PROGRAM ExtMode_Init
VAR
	iSTEP : INT:= 0;
	Pulse1			: TP; //for drive_on pulse
	Pulse2			: TP; //for ext_start pulse
	Pulse3			: TP;
	Pulse4			: TP;
	
	rInit			: R_TRIG;   // latch one press
	bInitLatch		: BOOL := FALSE;
	//bExtOK			: BOOL := IO_KUKA.bEXT_mode ;
	   
    rStep10       : R_TRIG;   // "step 10 entered" one-shot
    rStep30       : R_TRIG;   // "step 30 entered" one-shot
    tonPeri    : TON;      // wait for $PERI_RDY
    tonStart   : TON;      // wait for $PRO_ACT
    tPulse     : TIME := T#300MS;
    tPeriTO    : TIME := T#10S;
    tStartTO   : TIME := T#10S;
	
	
	
END_VAR


//// ================  Edges  ================
////rInit(CLK := IO_KUKA.Init_Cmd);
//rStep10(CLK := (iSTEP =10));
//rStep30(CLK := (iSTEP =30));

//IF IO_KUKA.Init_Cmd AND IO_KUKA.bEXT_mode = TRUE THEN
//	bInitLatch := TRUE;
//END_IF

//IF iSTEP <> 0 THEN
//	IO_control.bMove_enable := TRUE;   // $MOVE_ENABLE = 1
//    IO_control.bDrive_off   := FALSE;  // $DRIVES_OFF = 0
//	IO_control.bIO_Act      := TRUE;   // your "Activate interface" bit
//END_IF


//// ================  Machine state  ================
//CASE iSTEP OF
//	// ================  0 : idle  ================
//	0:	
//		IO_control.bDrive_on  	:= FALSE;
//  	 	IO_control.bExt_start 	:= FALSE;
//    	IO_control.bConf_msg  	:= FALSE;
//  		IO_control.bMove_enable := FALSE;
//    	IO_control.bIO_Act      := FALSE;
//   		IO_control.bDrive_off   := FALSE;
		
//		IF bInitLatch THEN
//			iSTEP := 10;
//		END_IF
		
//	// ================  10 : pulse drives_on, start wait for peri_rdy  ================
//	10:	
//		Pulse1(IN := rStep10.Q, PT := tPulse);
//		IO_control.bDrive_on := Pulse1.Q;
		
//		IF rStep10.Q THEN
//			tonPeri(IN := TRUE, PT := tPeriTO);
//			iSTEP := 20;
//		END_IF

		
//	// ================  20 : pwait for peri_rdy, conf_mess follows stopmess  ================
//	20:	
//		IO_control.bConf_msg := IO_KUKA.bStopmess;
		
//		IF IO_KUKA.bPeri_ready THEN
//			tonPeri(IN := FALSE);
//			iSTEP := 30;
//		ELSE
//			bInitLatch := FALSE;
//        	tonPeri(IN := FALSE);
//        	iSTEP := 0;
//		END_IF
	

//	// ================  30 : when no stopmess, pulse ext_start and wait Pro_act  ================
//	30:
//		IO_control.bConf_msg := IO_KUKA.bStopmess;
		
//		IF NOT IO_KUKA.bStopmess THEN
//			Pulse2(IN := rStep30.Q, PT := tPulse);
//			IO_control.bExt_start := Pulse2.Q;
			
//			IF rStep30.Q THEN
//				tonStart(IN := TRUE, PT := tStartTO);
//				iSTEP := 40;
//			END_IF
//		END_IF
		

//	// ================  40 : wait for pro_act, keep clearing stopmess ================
//	40:	
//		IO_control.bConf_msg := IO_KUKA.bStopmess;
		
//		IF IO_KUKA.bPro_act THEN
//			tonStart(IN := FALSE);
//			IO_control.bExt_start := FALSE;
//			bInitLatch := FALSE;
//			iSTEP := 0;
//		ELSIF tonStart.Q THEN
//			tonStart(IN := FALSE);
//			iSTEP := 30;	
//		END_IF
		
//ELSE
//	iSTEP := 0;		
		
//END_CASE




CASE iSTEP OF
	
	//KUKA ext init cmd
	0:	IF IO_KUKA.Init_Cmd THEN
			iSTEP := iSTEP + 1;
		END_IF
	
	//hardware toggle extmode n stopmess ON, then on move_enable n driveoff
	//then ON drive on
	1:	IF IO_KUKA.bEXT_mode THEN
			IO_KUKA.Init_Cmd := FALSE;
			IO_control.bMove_enable := IO_control.bDrive_off := TRUE;
			iSTEP := iSTEP + 1;
//		ELSE
//			IO_KUKA.Init_Cmd := FALSE;
//			iSTEP := 0;
		END_IF
		
	2:	IF IO_control.bMove_enable THEN
			IO_control.bIO_Act := TRUE;
			IO_control.bDrive_on := TRUE;
			IO_KUKA.Init_Cmd := FALSE;
			iSTEP := iSTEP + 1;
		END_IF	
	
	//if peri_ready on, then off drive_on
	3:	IF IO_KUKA.bPeri_ready THEN
			IO_control.bDrive_on := FALSE;
			iSTEP := iSTEP + 1;
		ELSE
			iSTEP := 0;
		END_IF
	
	//IF drive_on is ON, ON conf_mess, then if stopmess is OFF, OFF confmess
	4:	IF IO_control.bDrive_on = FALSE THEN
			IO_control.bConf_msg := TRUE;
			IF NOT IO_KUKA.bStopmess THEN
				IO_control.bConf_msg := FALSE;
				iSTEP := iSTEP + 1;
			ELSE
				iSTEP := 0;
			END_IF
		ELSE
			IO_KUKA.Init_Cmd := FALSE;
			iSTEP := 0;
		END_IF
	
	//confmess OFF, ON ext_start, when pro_act is OFF, off ext_start	
	5:	IF IO_control.bConf_msg = FALSE THEN
			IO_KUKA.bExt_start := TRUE;
			iSTEP := iSTEP + 1;
		ELSE
			iSTEP := 0;
		END_IF
		
	6:	IF IO_KUKA.bPro_act THEN
			IO_control.bExt_start := FALSE;		
			iSTEP := 0;
		ELSE
			iSTEP := 0;
		END_IF	
		
		
END_CASE

END_PROGRAM

(* stored: Version 1.1.0.1, ProductVersion 3.1.4024.12
   POU ExtMode_Init: Id {208ca540-6b2a-4ae5-84e7-ac901ada21d3}, SpecialFunc None *)
